// TIA Portal V17 program export: 1 tag tables, 0 data types, 1 data blocks, 1 code blocks (in call order from the OBs), 3 instance data blocks

VAR_GLOBAL   // PLC tag table "Default tag table"
   System_Byte AT %MB100 : Byte;
   FirstScan AT %M100.0 : Bool;
   DiagStatusUpdate AT %M100.1 : Bool;
   AlwaysTRUE AT %M100.2 : Bool;
   AlwaysFALSE AT %M100.3 : Bool;
   Clock_Byte AT %MB101 : Byte;
   Clock_10Hz AT %M101.0 : Bool;
   Clock_5Hz AT %M101.1 : Bool;
   "Clock_2.5Hz" AT %M101.2 : Bool;
   Clock_2Hz AT %M101.3 : Bool;
   "Clock_1.25Hz" AT %M101.4 : Bool;
   Clock_1Hz AT %M101.5 : Bool;
   "Clock_0.625Hz" AT %M101.6 : Bool;
   "Clock_0.5Hz" AT %M101.7 : Bool;
   M_CurrentDateTimeStatus AT %MW166 : Int;
END_VAR

DATA_BLOCK "DB - 1 - Dados Inversor MB-01"   // DB230
{ S7_Optimized_Access := 'FALSE' }
VERSION : 0.1
// stored: AutoNumber false, IsOnlyStoredInLoadMemory false, IsWriteProtectedInAS false
   VAR RETAIN
      RW_TCPModBUS_IP_Oct_1_MB : USInt := 0;   // IP Octeto 1 do Inversor MB
      RW_TCPModBUS_IP_Oct_2_MB : USInt := 0;   // IP Octeto 2 do Inversor MB
      RW_TCPModBUS_IP_Oct_3_MB : USInt := 0;   // IP Octeto 3 do Inversor MB
      RW_TCPModBUS_IP_Oct_4_MB : USInt := 0;   // IP Octeto 4 do Inversor MB
      RW_MinMotorFreqHz_MB_Hz : UInt := 300;   // Frequência Minima do Motor Utilizado para o controle de velocidade
      RW_MaxMotorFreqHz_MB_Hz : UInt := 600;   // Frequência Máxima do Motor
      RO_SomatorioConsumo_kWh { ExternalAccessible := 'False'; ExternalVisible := 'False'; ExternalWritable := 'False'} : Real;
      RO_CorrenteAtual_A { ExternalAccessible := 'False'; ExternalVisible := 'False'; ExternalWritable := 'False'} : Real;
      RO_FrequenciaAtual_Hz { ExternalAccessible := 'False'; ExternalVisible := 'False'; ExternalWritable := 'False'} : Real;
      RO_PotenciaAtual_kW { ExternalAccessible := 'False'; ExternalVisible := 'False'; ExternalWritable := 'False'} : Real;
      RO_TensaoAtualSaida_V { ExternalVisible := 'False'} : Real;
      RO_MotorRPM { ExternalAccessible := 'False'; ExternalVisible := 'False'; ExternalWritable := 'False'} : Real;
      RO_TempDriveDissipadorCalor_C { ExternalAccessible := 'False'; ExternalVisible := 'False'; ExternalWritable := 'False'} : Real;
      RO_TempDriveCartaoControle_C { ExternalAccessible := 'False'; ExternalVisible := 'False'; ExternalWritable := 'False'} : Real;
      RO_HorimetroMotor_H : Real;
      RO_HorimetroDrive_H : Real;
      RO_UltimoAlarme : Int;
      "RO_AnalogInput53_ma-V" : Real;
      "RO_AnalogInput54_ma-V" : Real;
      Cfg_Potencia_Motor_kW : Real;
      Cfg_Motor_hp : Real;
      Cfg_Motor_TensaoNominal_V : Real;
      Cfg_Corrente_Nominal_A : Real;
      Cfg_Velocidade_Nominal_RPM : Real;
      RO_Numero_de_PartidasMotor : Real;
      RO_Numero_de_PartidasDrive : Real;
      RO_TensaoBarramentoDC_V : Real;
      RO_TensaoAmpla_V : Real;
   END_VAR
BEGIN
END_DATA_BLOCK

ORGANIZATION_BLOCK "Main"   // OB1, LAD, ProgramCycle
TITLE = "Main Program Sweep (Cycle)"
{ S7_Optimized_Access := 'TRUE' }
VERSION : 0.1
// stored: AutoNumber true, IsIECCheckEnabled false, SetENOAutomatically false
BEGIN

REGION Network 1: Operations
END_REGION

REGION Network 2: Root
END_REGION
END_ORGANIZATION_BLOCK

DATA_BLOCK "DB - 1 - Modbus Danfoss - MB-01"   // DB7
// stored: AutoNumber true, InstanceOfName FB - 1 - Modbus Danfoss - MB-01, InstanceOfType FB
"FB - 1 - Modbus Danfoss - MB-01"
   // VAR_INPUT
   //    FirstScan : Bool;
   //    RW_TCPModBUS_IP_Oct_1_MB : USInt;
   //    RW_TCPModBUS_IP_Oct_2_MB : USInt;
   //    RW_TCPModBUS_IP_Oct_3_MB : USInt;
   //    RW_TCPModBUS_IP_Oct_4_MB : USInt;
   //    RW_MinMotorFreqHz_MB_Hz : UInt;
   //    RW_MaxMotorFreqHz_MB_Hz : UInt;
   // END_VAR
   // VAR_OUTPUT
   //    RO_SomatorioConsumo_kWh : Real;
   //    RO_CorrenteAtual_A : Real;
   //    RO_FrequenciaAtual_Hz : Real;
   //    RO_PotenciaAtual_kW : Real;
   //    RO_TensaoAtualSaida_V : Real;
   //    RO_MotorRPM : Real;
   //    RO_TempDriveDissipadorCalor_C : Real;
   //    RO_TempDriveCartaoControle_C : Real;
   //    RO_HorimetroMotor_H : Real;
   //    RO_HorimetroDrive_H : Real;
   //    RO_UltimoAlarme : Int;
   //    "RO_AnalogInput53_ma-V" : Real;
   //    "RO_AnalogInput54_ma-V" : Real;
   //    Cfg_Potencia_Motor_kW : Real;
   //    Cfg_Motor_hp : Real;
   //    Cfg_Motor_TensaoNominal_V : Real;
   //    Cfg_Corrente_Nominal_A : Real;
   //    Cfg_Velocidade_Nominal_RPM : Real;
   //    RO_Numero_de_PartidasMotor : Real;
   //    RO_Numero_de_PartidasDrive : Real;
   //    RO_TensaoBarramento_DC_V : Real;
   //    RO_TensaoAmpla_V : Real;
   // END_VAR
   // VAR
   //    MB_Mode { ExternalAccessible := 'False'; ExternalVisible := 'False'; ExternalWritable := 'False'} : USInt;
   //    DataLen { ExternalAccessible := 'False'; ExternalVisible := 'False'; ExternalWritable := 'False'} : USInt;
   //    tmp_real { ExternalAccessible := 'False'; ExternalVisible := 'False'; ExternalWritable := 'False'} : Real;
   //    tmp_word { ExternalAccessible := 'False'; ExternalVisible := 'False'; ExternalWritable := 'False'} : Word;
   //    M_DataAddrReq { ExternalAccessible := 'False'; ExternalVisible := 'False'; ExternalWritable := 'False'} : UDInt;
   //    TypeWrite { ExternalAccessible := 'False'; ExternalVisible := 'False'; ExternalWritable := 'False'} : Bool;
   //    Alternate { ExternalAccessible := 'False'; ExternalVisible := 'False'; ExternalWritable := 'False'} : Int;
   //    M_TCPTmpValueDWord { ExternalAccessible := 'False'; ExternalVisible := 'False'; ExternalWritable := 'False'} : DWord;
   //    M_TCPTmpValueUInt { ExternalAccessible := 'False'; ExternalVisible := 'False'; ExternalWritable := 'False'} : UInt;
   // END_VAR
BEGIN
END_DATA_BLOCK

DATA_BLOCK "MB_CLIENT_Inv01"   // DB22
// stored: AutoNumber false, InstanceOfName MB_CLIENT, OfSystemLibElement MB_CLIENT, OfSystemLibVersion 2.0
"MB_CLIENT"
   // VAR_INPUT
   //    REQ : Bool;
   //    DISCONNECT : Bool;
   //    CONNECT_ID : UInt;
   //    IP_OCTET_1 : USInt;
   //    IP_OCTET_2 : USInt;
   //    IP_OCTET_3 : USInt;
   //    IP_OCTET_4 : USInt;
   //    IP_PORT : UInt;
   //    MB_MODE : USInt;
   //    MB_DATA_ADDR : UDInt;
   //    MB_DATA_LEN : UInt;
   // END_VAR
   // VAR_OUTPUT
   //    DONE : Bool;
   //    BUSY : Bool;
   //    ERROR : Bool;
   //    STATUS : Word;
   // END_VAR
   // VAR_IN_OUT
   //    MB_DATA_PTR : Variant;
   // END_VAR
   // VAR
   //    TCON_SFB { S7_SetPoint := 'True'} : TCON;
   //    TDISCON_SFB { S7_SetPoint := 'True'} : TDISCON;
   //    TSEND_SFB { S7_SetPoint := 'True'} : TSEND;
   //    TRCV_SFB { S7_SetPoint := 'True'} : TRCV;
   //    TCON_PARAM { S7_SetPoint := 'True'} : TCON_Param;
   //    PF_FREQUENCY : Real;
   //    BLOCKED_PROC_TIMEOUT : Real;
   //    RCV_TIMEOUT : Real;
   //    CURRENT_TIME_VALUE : DWord;
   //    SAVED_TIME_VALUE : DWord;
   //    XMT_TIME : DWord;
   //    SAVED_CONNECT_ID : Word;
   //    SAVED_IP_PORT : Word;
   //    SAVED_MODE : Byte;
   //    SAVED_IP1 : Byte;
   //    SAVED_IP2 : Byte;
   //    SAVED_IP3 : Byte;
   //    SAVED_IP4 : Byte;
   //    SAVED_DATA_ADDR : DWord;
   //    SAVED_DATA_LEN : Word;
   //    MB_STATE : Word;
   //    COMM_SENT_COUNT : Word;
   //    BYTE_COUNT : Word;
   //    BYTE_COUNTB : Byte;
   //    SAVED_START_ADDR : Word;
   //    MB_TRANSACTION_ID : Word;
   //    MB_UNIT_ID : Word;
   //    RETRIES : Word;
   //    INIT_OK : Bool;
   //    ACTIVE : Bool;
   //    CONNECTED : Bool;
   //    SAVED_MA_REQ : Bool;
   // END_VAR
BEGIN
END_DATA_BLOCK

DATA_BLOCK "T_Alternate_1"   // DB20
{ S7_Optimized_Access := 'TRUE' }
// stored: AutoNumber true, InstanceOfName IEC_TIMER, OfSystemLibElement IEC_TIMER, OfSystemLibVersion 1.0
"IEC_TIMER"
   // VAR
   //    PT : Time;
   //    ET { ExternalWritable := 'False'} : Time;
   //    IN : Bool;
   //    Q { ExternalWritable := 'False'} : Bool;
   // END_VAR
BEGIN
END_DATA_BLOCK
